Universal Robots PolyScope program: 20250522.urp

Program 20250522 (installation=20240827 directory=/programs/con createdIn=5.15.1 lastSavedIn=5.15.1 robotSerialNumber=20245500285)
Calibrated DH parameters: a=[0.000097, -0.210459, -0.026602, 0.000137, 0.000078, 0]; d=[0.162601, 254.180657, -54.076236, -199.970743, 0.099615, 0.099684]; alpha=[1.569796, -0.001455, 0.001957, 1.570525, -1.571561, 0]; deltaTheta=[0, -1.053331, 8.839472, -1.50296, 0.000002, 0]
InitVariablesNode
Robot Program (runOnlyOnce=false)
  MoveJ speed 60 deg/s, acceleration 80 deg/s^2 (useActiveTCP=true) feature=Base
    Waypoint goudo: motionParameters(jointSpeed=1.047198 jointAcceleration=1.396263 cartesianSpeed=0.25 cartesianAcceleration=1.2); TCP in base x=804.816 y=122.737 z=261.364 mm, rx=1.21 ry=1.2107 rz=1.2121 rad; joints [178.646, -48.519, 103.06, -234.54, -88.651, 180.01] deg; TCP offset x=-0.17 y=0 z=192.95 mm, rx=0 ry=0 rz=0 rad
    Popup Message (haltProgram=false message=tcp inputType=Text)
    Waypoint tcp: TCP in base x=804.824 y=122.726 z=254.616 mm, rx=1.21 ry=1.2106 rz=1.2122 rad; joints [178.644, -47.754, 103.049, -235.296, -88.65, 180.008] deg
    x := 0.006
    y := 0.006
    z := 0.001
    a1 := p[0,0,-z*1,0,0,0]
    a2 := p[0,0,-z*2,0,0,0]
    a3 := p[0,0,-z*3,0,0,0]
    b1 := p[x,y,-z*1,0,0,0]
    b2 := p[x,y,-z*2,0,0,0]
    b3 := p[x,y,-z*3,0,0,0]
    c1 := p[-x,y,-z*1,0,0,0]
    c2 := p[-x,y,-z*2,0,0,0]
    c3 := p[-x,y,-z*3,0,0,0]
    d1 := p[-x,-y,-z*1,0,0,0]
    d2 := p[-x,-y,-z*2,0,0,0]
    d3 := p[-x,-y,-z*3,0,0,0]
    e1 := p[x,-y,-z*1,0,0,0]
    e2 := p[x,-y,-z*2,0,0,0]
    e3 := p[x,-y,-z*3,0,0,0]
    tcpa1 := pose_add(tcp, a1)
    tcpa2 := pose_add(tcp, a2)
    tcpa3 := pose_add(tcp, a3)
    tcpb1 := pose_add(tcp, b1)
    tcpb2 := pose_add(tcp, b2)
    tcpb3 := pose_add(tcp, b3)
    tcpc1 := pose_add(tcp, c1)
    tcpc2 := pose_add(tcp, c2)
    tcpc3 := pose_add(tcp, c3)
    tcpd1 := pose_add(tcp, d1)
    tcpd2 := pose_add(tcp, d2)
    tcpd3 := pose_add(tcp, d3)
    tcpe1 := pose_add(tcp, e1)
    tcpe2 := pose_add(tcp, e2)
    tcpe3 := pose_add(tcp, e3)
    MoveJ speed 60 deg/s, acceleration 80 deg/s^2 (useActiveTCP=true) feature=Base
      Popup Message (haltProgram=false message=az1 inputType=Text)
      Waypoint Variable (Variable): variable=tcpa1
      Popup Message (haltProgram=false message=az2 inputType=Text)
      Waypoint Variable (Variable): variable=tcpa2
      Popup Message (haltProgram=false message=az3 inputType=Text)
      Waypoint Variable (Variable): variable=tcpa3
      Popup Message (haltProgram=false message=guodu inputType=Text)
      Waypoint goudo: TCP in base x=804.816 y=122.737 z=261.364 mm, rx=1.21 ry=1.2107 rz=1.2121 rad; joints [178.646, -48.519, 103.06, -234.54, -88.651, 180.01] deg
      Popup Message (haltProgram=false message=bz1 inputType=Text)
      Waypoint Variable (Variable): variable=tcpb1
      Popup Message (haltProgram=false message=bz2 inputType=Text)
      Waypoint Variable (Variable): variable=tcpb2
      Popup Message (haltProgram=false message=bz3 inputType=Text)
      Waypoint Variable (Variable): variable=tcpb3
      Popup Message (haltProgram=false message=guodu inputType=Text)
      Waypoint goudo: TCP in base x=804.816 y=122.737 z=261.364 mm, rx=1.21 ry=1.2107 rz=1.2121 rad; joints [178.646, -48.519, 103.06, -234.54, -88.651, 180.01] deg
      Popup Message (haltProgram=false message=cz1 inputType=Text)
      Waypoint Variable (Variable): variable=tcpc1
      Popup Message (haltProgram=false message=cz2 inputType=Text)
      Waypoint Variable (Variable): variable=tcpc2
      Popup Message (haltProgram=false message=cz3 inputType=Text)
      Waypoint Variable (Variable): variable=tcpc3
      Popup Message (haltProgram=false message=guodu inputType=Text)
      Waypoint goudo: TCP in base x=804.816 y=122.737 z=261.364 mm, rx=1.21 ry=1.2107 rz=1.2121 rad; joints [178.646, -48.519, 103.06, -234.54, -88.651, 180.01] deg
      Popup Message (haltProgram=false message=dz1 inputType=Text)
      Waypoint Variable (Variable): variable=tcpd1
      Popup Message (haltProgram=false message=dz2 inputType=Text)
      Waypoint Variable (Variable): variable=tcpd2
      Popup Message (haltProgram=false message=dz3 inputType=Text)
      Waypoint Variable (Variable): variable=tcpd3
      Popup Message (haltProgram=false message=guodu inputType=Text)
      Waypoint goudo: TCP in base x=804.816 y=122.737 z=261.364 mm, rx=1.21 ry=1.2107 rz=1.2121 rad; joints [178.646, -48.519, 103.06, -234.54, -88.651, 180.01] deg
      Popup Message (haltProgram=false message=ez1 inputType=Text)
      Waypoint Variable (Variable): variable=tcpe1
      Popup Message (haltProgram=false message=ez2 inputType=Text)
      Waypoint Variable (Variable): variable=tcpe2
      Popup Message (haltProgram=false message=ez3 inputType=Text)
      Waypoint Variable (Variable): variable=tcpe3
      Popup Message (haltProgram=false message=guodu inputType=Text)
